Staubli VAL3: SUB.dtx

num nChar = 89
num nFile = 2
num nPath
public string sItems
string sSession
progItem pEdit
  [0]
    InstrItem iEvent
      [0]
        string sType
        string sData
    string sID
num nKey
